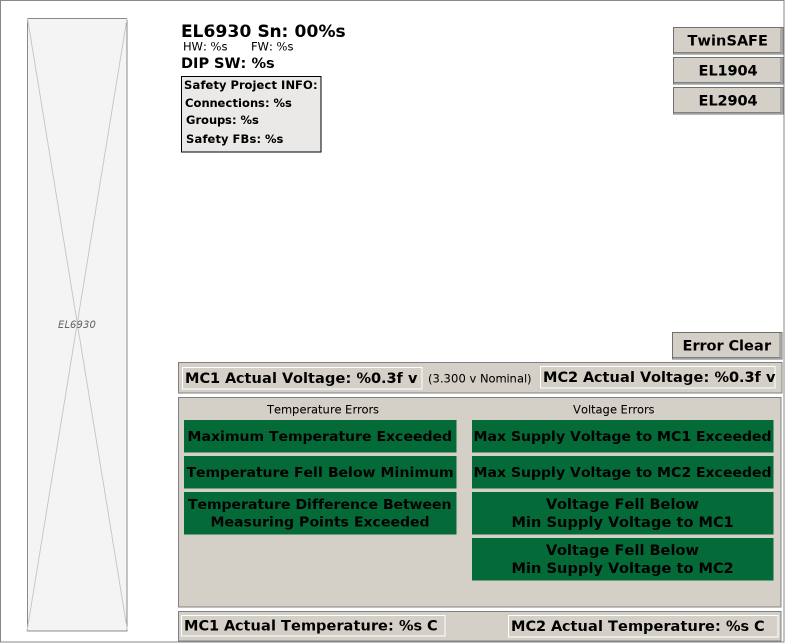
VISUALIZATION EL6930_Specific_Diagnostics  // 785x643
    Button (673,27 110x27), "TwinSAFE"
        OnMouseClick: change screen: TwinSAFE
    Button (673,57 110x27), "EL1904"
        OnMouseClick: change screen: EL1904_Specific_Diagnostics
    Button (673,87 110x27), "EL2904"
        OnMouseClick: change screen: EL2904_Specific_Diagnostics
    Rectangle (178,20 275x22), "EL6930 Sn: 00%s", text variable: g_dwHMI_EL6930Sn
    Rectangle (180,38 65x17), "HW: %s", text variable: g_sHMI_EL6930_HWvers
    Rectangle (248,38 65x17), "FW: %s", text variable: g_sHMI_EL6930_FWvers
    Rectangle (178,52 164x22), "DIP SW: %s", text variable: g_wHMI_EL6930DSw
    Group (181,74 140x78)
        Rectangle (0,2 140x76)
        Rectangle (1,17 135x24), "Connections: %s", text variable: g_bHMI_EL6930_NoOfConnections
        Label (0,0 135x22), "Safety Project INFO:"
        Rectangle (2,34 135x24), "Groups: %s", text variable: g_bHMI_EL6930_NoOfSafetyGrps
        Rectangle (2,53 135x24), "Safety FBs: %s", text variable: g_bHMI_EL6930_NoOfSafetyFBs
    Button (672,332 110x27), "Error Clear"
        OnMouseUp: execute { g_xHMI_EL6930_ErrClearPB := FALSE ; }
        OnMouseDown: execute { g_xHMI_EL6930_ErrClearPB := TRUE ; }
    Group (178,362 604x31)
        Rectangle (0,0 604x31)
        Label (243,9 118x15), "(3.300 v Nominal)"
        Rectangle (4,5 240x22), "MC1 Actual Voltage: %0.3f v", text variable: g_wHMI_EL6930PriMC_Volts
        Rectangle (362,4 235x22), "MC2 Actual Voltage: %0.3f v", text variable: g_wHMI_EL6930SecMC_Volts
    Group (178,611 603x30)
        Rectangle (0,0 603x30)
        Rectangle (3,4 264x21), "MC1 Actual Temperature: %s C", text variable: g_wHMI_EL6930PriMCTemp
        Rectangle (330,4 270x22), "MC2 Actual Temperature: %s C", text variable: g_wHMI_EL6930SecMCTemp
    Group (178,397 603x210)
        Rectangle (0,0 603x210)
        Label (80,0 130x25), "Temperature Errors"
        Rectangle (6,23 272x32), "Maximum Temperature Exceeded", colour toggle: g_xHMI_EL6930_MaxTemp
        Label (371,0 130x25), "Voltage Errors"
        Rectangle (6,59 272x32), "Temperature Fell Below Minimum", colour toggle: g_xHMI_EL6930_MinTemp
        Rectangle (6,95 272x42), "Temperature Difference Between Measuring Points Exceeded", colour toggle: g_xHMI_EL6930_TempDiffExceeded
        Rectangle (294,23 301x32), "Max Supply Voltage to MC1 Exceeded", colour toggle: g_xHMI_EL6930_MaxVccMC1
        Rectangle (294,59 301x32), "Max Supply Voltage to MC2 Exceeded", colour toggle: g_xHMI_EL6930_MaxVccMC2
        Rectangle (294,95 301x42), "Voltage Fell Below Min Supply Voltage to MC1", colour toggle: g_xHMI_EL6930_MinVccMC1
        Rectangle (294,141 301x42), "Voltage Fell Below Min Supply Voltage to MC2", colour toggle: g_xHMI_EL6930_MinVccMC2
    Image (27,18 100x613), image: EL6930
END_VISUALIZATION

(* stored: Version 1.1.0.1, ProductVersion 3.1.0.18
   Visu EL6930_Specific_Diagnostics: Id {06f67e71-55a0-4de4-a6e2-35dfd574a88f} *)
